INTERFACE ITF_CUSTOM_SKILL

PROPERTY Operational : BOOL
SET
END_SET
END_PROPERTY

{warning 'Add method implementation '}
METHOD StartCustomSkill : eResult
END_METHOD

{warning 'Add method implementation '}
METHOD StopCustomSkill : eResult
END_METHOD

END_INTERFACE

(* stored: Version 1.1.0.1, ProductVersion 3.1.4026.18
   Itf ITF_CUSTOM_SKILL: Id {8f6eace4-1ce3-47c4-ac9d-cfdc087b1091}
   Folder incl Call Parent: Id {3fd66bbc-28bb-4062-b165-021c15079841}
   Property Operational: Id {8dbad60b-2af7-4d53-8ea7-bd74c989b93d}
   Set Set: Id {c0a0151e-b8e4-45d3-9ae4-094595e63945}
   Method StartCustomSkill: Id {e26c5811-9a9c-41cd-a3f6-36e61b48ba59}
   Method StopCustomSkill: Id {f6f30784-7f29-4946-b6ca-b0a6d6572b85} *)
